RoboDK station: New Station.rdk

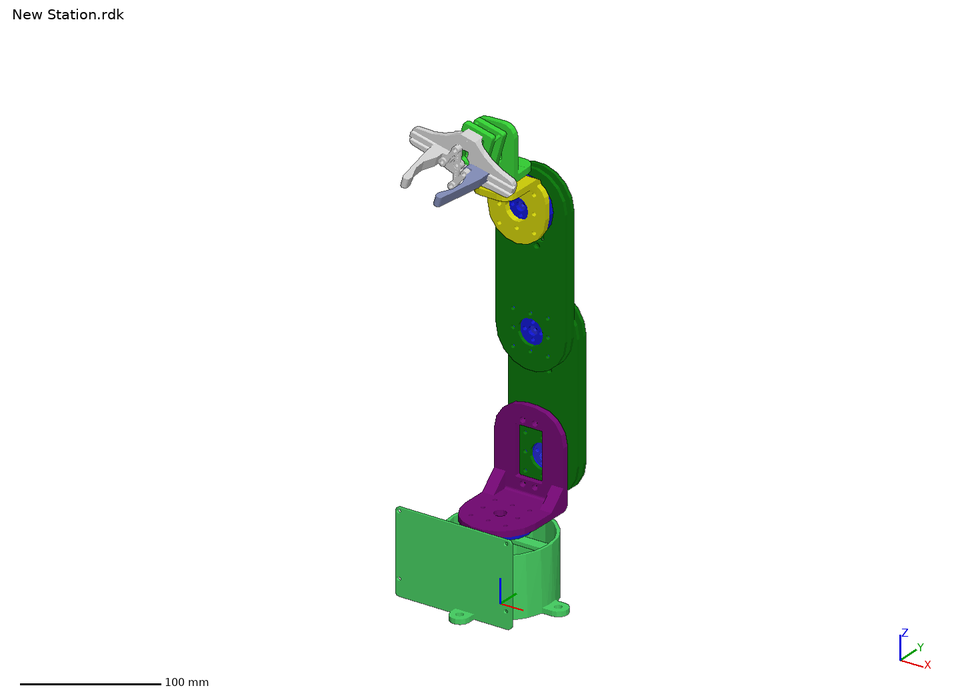
[picture v0: the station drawn from its stored meshes, robots at their saved joint values, targets as dots, program paths as lines]
Station New Station (saved by RoboDK 5.6.8). Poses are relative to the parent item; angles as X-Y-Z fixed-axis rotations.
  - frame Frame 2 at (0, 0, 0) mm
    - object main2 at (0, 0, 0) mm, geometry from main2.STEP
      - item type 7 Base
      - item type 7 
      - item type 7 Shoulder
      - item type 7 Elbow
      - item type 7 Wrist1
      - item type 7 Wrist2
      - item type 7 
      - item type 7 EE
  - frame My Robot Frame at (0, 0, 0) mm
    - robot My Robot: 6 axes
        modified DH rows (alpha deg, a mm, theta deg, d mm): 0, 0, 90, 94.85; 90, 0, 90, 0; 0, 104, 0, 0; 0, 104, -90, 0; -90, 0, 0, 66.6; 90, 0, 0, 58.95
        joint limits [0, -90, -90, -90, -90, -90] to [180, 90, 90, 90, 90, 90]; home [90, 0, 0, 0, 0, 0]; saved at [90, 0, 0, 0, -3.51, 15.78]
